PROGRAM Main_SendData
VAR	
	Done		: BOOL;
	Sent		: BOOL;
	New_Data	: BOOL;
	Saved		: BOOL;
END_VAR

(* get data from database *)
Get_Data();
 
IF New_Data := Get_Data.Done THEN
	(* send data to aws iot core *)
	IF NOT Sent THEN
		Send_Data();
		
		IF Send_Data.Published THEN
			Sent	:= TRUE;
		END_IF	
		
	END_IF
	
	(* save data to localdb *)
	IF Sent THEN
		Save_Data();
		
		IF Save_Data.Done THEN
			Saved := TRUE;
		END_IF	
		
	END_IF
	
ELSE
	Sent	:= FALSE;
	Saved 	:= FALSE;
	
END_IF

END_PROGRAM

(* stored: Version 1.1.0.1, ProductVersion 3.1.4024.6
   POU Main_SendData: Id {f159ed40-cca9-4e3d-ac6a-ec5e9cf1af8e}, SpecialFunc None *)
